FUNCTION_BLOCK FB_4_InsertarBasePale_SFCC
VAR_INPUT

	//  SFC-Flags
	SFCPause: BOOL;
	SFCReset: BOOL;

	// Indicadores de sincronización
	Ack: BOOL := TRUE;
	Execute: BOOL;
	
	// Entradas
	VerticalArriba: BOOL;
	VerticalAbajo: BOOL;
	VacioDescargador: BOOL;	
	DescargadorDetras: BOOL;
	DescargadorDelante: BOOL;
	
END_VAR
VAR_OUTPUT
	
// Indicadores de sincronización
	Ready: BOOL;	
	Done: BOOL;
	
	// Salidas
	DescargadorAtras: BOOL;
	DescargadorAdelante: BOOL;
	DescargadorBaja : BOOL;
	EyectorSucciona : BOOL;
	
END_VAR
VAR
END_VAR

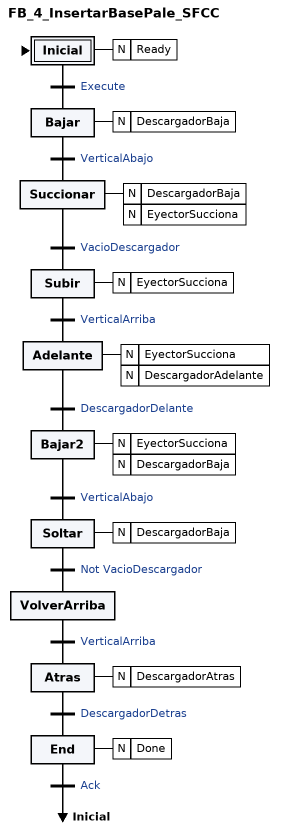
INITIAL_STEP Inicial:
    Ready(N);
END_STEP
TRANSITION FROM Inicial TO Bajar
    := Execute;
END_TRANSITION
STEP Bajar:
    DescargadorBaja(N);
END_STEP
TRANSITION FROM Bajar TO Succionar
    := VerticalAbajo;
END_TRANSITION
STEP Succionar:
    DescargadorBaja(N);
    EyectorSucciona(N);
END_STEP
TRANSITION FROM Succionar TO Subir
    := VacioDescargador;
END_TRANSITION
STEP Subir:
    EyectorSucciona(N);
END_STEP
TRANSITION FROM Subir TO Adelante
    := VerticalArriba;
END_TRANSITION
STEP Adelante:
    EyectorSucciona(N);
    DescargadorAdelante(N);
END_STEP
TRANSITION FROM Adelante TO Bajar2
    := DescargadorDelante;
END_TRANSITION
STEP Bajar2:
    EyectorSucciona(N);
    DescargadorBaja(N);
END_STEP
TRANSITION FROM Bajar2 TO Soltar
    := VerticalAbajo;
END_TRANSITION
STEP Soltar:
    DescargadorBaja(N);
END_STEP
TRANSITION FROM Soltar TO VolverArriba
    := Not VacioDescargador;
END_TRANSITION
STEP VolverArriba:
END_STEP
TRANSITION FROM VolverArriba TO Atras
    := VerticalArriba;
END_TRANSITION
STEP Atras:
    DescargadorAtras(N);
END_STEP
TRANSITION FROM Atras TO End
    := DescargadorDetras;
END_TRANSITION
STEP End:
    Done(N);
END_STEP
TRANSITION FROM End TO Inicial
    := Ack;
END_TRANSITION

END_FUNCTION_BLOCK

(* stored: Version 1.1.0.1, ProductVersion 3.1.4024.12
   POU FB_4_InsertarBasePale_SFCC: Id {baeb7dee-dd04-40cf-8851-aefbd46ea0d7}, SpecialFunc None *)
